(*********************************** G.D S.p.A. - Technical Department ***********************************
============= PROGRAM INFO ============
FOLDER:             TBD
MACHINES INVOLVED:  TBD 

============= DESCRIPTION =============
csp machine declaration

============= REVISIONS ===============
Date		Version	 	Author      	Description             
----------	-------		------------  	--------------------------------------------
2019/04/05 	0000.00	 	M.Grasso		Creation of the PRG

**********************************************************************************************************)
(*$R process_ref := prc; $*)
PROGRAM csp_case_glue_os_accU
VAR
	
	prc:											process;
	prc_path:										STRING;
END_VAR

_read_var_input();

_object_manager();

IF NOT objects_running()
THEN
	RETURN;	
END_IF

_read_process_image();

_mode_manager();

_set_runtime_properties();

(********************************* BODY *********************************)
(************************************************************************)

_handle_messages();

_write_output();

ACTION _handle_messages:
;
END_ACTION

ACTION _handle_process_test:
;
END_ACTION

ACTION _mode_manager:
IF process_mode_req_is_pending(prc)
THEN
    process_apply_mode_req_first_step(prc);
    CASE process_get_mode(prc) OF
        MODE_TO_ABSENT:
			;
        MODE_TO_INACTIVE:
			;
        MODE_TO_TEST:
			;
        MODE_TO_OPERATIONAL:
			;
    END_CASE
    process_apply_mode_req_second_step(prc);
END_IF
END_ACTION

ACTION _object_manager:
IF objects_initialization()
THEN
	sub_process_init(
		object_name					:= 'csp_case_glue_os_accU.prc', 
		process						:= csp_case_glue_os.prc, 
		CONVERSION_this				:= prc);
		
	prc_path 						:= process_get_path(prc);
END_IF

IF objects_running()
THEN
	process_cycle(prc);
END_IF
END_ACTION

ACTION _read_process_image:
;
END_ACTION

ACTION _read_var_input:
;
END_ACTION

ACTION _set_runtime_properties:
;
END_ACTION

ACTION _write_output:
;
END_ACTION

END_PROGRAM

(* stored: Version 1.1.0.1, ProductVersion 3.1.4022.12
   POU csp_case_glue_os_accU: Id {9a7dd4e0-5673-4b8c-9647-5d1eb80dde82}, SpecialFunc None
   Action _handle_messages: Id {afa77949-af31-44ec-838d-b8ab80a0950e}
   Action _handle_process_test: Id {2ad43e13-8395-4a01-997c-d9926fd604ed}
   Action _mode_manager: Id {a27e0a0e-bf21-4eb6-be36-250ef573573f}
   Action _object_manager: Id {52814d8b-6038-425c-a911-642b1339f9a4}
   Action _read_process_image: Id {bb937d64-7a0c-4ba1-9fad-70b4491247e5}
   Action _read_var_input: Id {b49327e9-7728-4950-b831-bed255a71a64}
   Action _set_runtime_properties: Id {f4f9beb7-6804-4050-a95f-3c4c312030db}
   Action _write_output: Id {0258d6ee-97b8-455e-b236-ac810a7dbafd} *)
